// TwinCAT 3 PLC project PLC
// ProgramVersion: 3.1.4024.0
// libraries:
//   Tc2_Standard, * (Beckhoff Automation GmbH)
//   Tc2_System, * (Beckhoff Automation GmbH)
//   Tc3_Module, * (Beckhoff Automation GmbH)
//   Util, * (System)
// project tree:
//   Diagnostic/ GVL_Diagnostic.TcGVL, ST_Diagnostic.TcDUT
//   FLM/Corking/ FB_CorkingRotation.TcPOU, E_FLM_CorkingStep.TcDUT, FB_FLM_CorkingStateMachine.TcPOU, ST_FLM_CorkingParams.TcDUT, ST_FLM_CorkingStatus.TcDUT
//   FLM/Enums/ E_FLM_Step.TcDUT
//   FLM/FBs/ FB_FLM_Diagnostic.TcPOU, FB_FLM_ReadCmd.TcPOU, FB_FLM_ReadCtrl.TcPOU, FB_FLM_ReadInputs.TcPOU, FB_FLM_ResetCmd.TcPOU, FB_FLM_WriteOutputs.TcPOU, FB_FLM_StateMachine.TcPOU
//   FLM/ FB_FLM_Main.TcPOU
//   FLM/Functions/ F_FLM_RawToLevel.TcPOU
//   FLM/Structs/ ST_FLM_Cmd.TcDUT, ST_FLM_Ctrl.TcDUT, ST_FLM_In.TcDUT, ST_FLM_Motion.TcDUT, ST_FLM_Out.TcDUT, ST_FLM_Params.TcDUT, ST_FLM_RawIn.TcDUT, ST_FLM_RawOut.TcDUT, ST_FLM_Status.TcDUT, ST_FLM_StatusSaved.TcDUT
//   / GlobalTextList.TcGTLO, PlcTask.TcTTO, SimuTask.TcTTO, VisualizationManager.TcVMO (not stored)
//   GVLs/ GVL_PLC.TcGVL
//   POUs/ PLC_MAIN.TcPOU, SIMU_MAIN.TcPOU
//   Simulation/ FB_VisuSim.TcPOU
//   StateMachinePro/ E_Step.TcDUT, FB_StateMachinePro.TcPOU
//   StateMachine/ FB_StateMachine.TcPOU
//   VISUs/ Visu.TcVIS
// real-time tasks:
//   TASK PlcTask: cycle T#10ms, priority 20, ADS port 350
//   TASK VISU_TASK: cycle T#200000us, priority 30, ADS port 351
//   TASK SimuTask: cycle T#10ms, priority 21, ADS port 352

CONFIGURATION PLC
    RESOURCE PLC ON TwinCAT3
        TASK PlcTask(INTERVAL := T#10ms, PRIORITY := 20);
        TASK SimuTask(INTERVAL := T#10ms, PRIORITY := 21);
        PROGRAM PLC_MAIN WITH PlcTask : PLC_MAIN;
        PROGRAM SIMU_MAIN WITH SimuTask : SIMU_MAIN;
    END_RESOURCE
END_CONFIGURATION

// ---- Diagnostic/ST_Diagnostic.TcDUT
(* -----------------------------------------------------------------------------
| This sample has been supplied by Beckhoff As-Is and is intended only as an   |
| example implementation. Functionality is not guaranteed.                     |
----------------------------------------------------------------------------- *)

TYPE ST_Diagnostic :
STRUCT
	aCritical : ARRAY[0..GVL_Diagnostic.cMAXEVENTS - 1] OF BOOL;	// eventi critici
	aError : ARRAY[0..GVL_Diagnostic.cMAXEVENTS - 1] OF BOOL;		// errori
	aWarning : ARRAY[0..GVL_Diagnostic.cMAXEVENTS - 1] OF BOOL;		// segnalazioni
	aInfo : ARRAY[0..GVL_Diagnostic.cMAXEVENTS - 1] OF BOOL;		// informazioni
	aVerbose : ARRAY[0..GVL_Diagnostic.cMAXEVENTS - 1] OF BOOL;		// messaggi
END_STRUCT
END_TYPE

// ---- FLM/Enums/E_FLM_Step.TcDUT
(* -----------------------------------------------------------------------------
| This sample has been supplied by Beckhoff As-Is and is intended only as an   |
| example implementation. Functionality is not guaranteed.                     |
----------------------------------------------------------------------------- *)

{attribute 'qualified_only'}
{attribute 'strict'}
{attribute 'to_string'}

TYPE E_FLM_Step :
(
	(* special steps *)
	NoStep := -32767,		// nessuno step
	Unknown := -32000,		// step sconosciuto
	
	(* Error steps *)
	NeOrError := -990,		// non abilitata o in errore
	Reset := -980,			// azzeramento errori

	(* Stop *)
	Stop := 0,				// stop
	
	(* Cycle *)
	Feeding := 110,			// avanzamento
	WaterFilling := 120,	// riempimento acqua
	MintFilling := 130,		// riempimento menta
	Corking := 150,			// tappatura	
		
	(* Stopping *)
	Stopping := 900
	
);
END_TYPE

// ---- FLM/Corking/E_FLM_CorkingStep.TcDUT
(* -----------------------------------------------------------------------------
| This sample has been supplied by Beckhoff As-Is and is intended only as an   |
| example implementation. Functionality is not guaranteed.                     |
----------------------------------------------------------------------------- *)

{attribute 'qualified_only'}
{attribute 'strict'}
{attribute 'to_string'}

TYPE E_FLM_CorkingStep :
(
	(* special steps *)
	NoStep := -32767,		// nessuno step
	Unknown := -32000,		// step sconosciuto
	
	(* Error steps *)
	NeOrError := -990,		// non abilitata o in errore
	Reset := -980,			// azzeramento errori
		
	(* Stop *)
	Stop := 0,
	
	(* Ready *)
	Ready := 100,	
	
	(* Cycle *)
	Down := 200,			// movimento verticale verso il basso
	Rotation := 210,		// rotazione 
	Up := 220,				// movimento verticale verso l'alto
	Done := 230,			// ciclo concluso
	(* Stopping *)
	Stopping := 900	
);
END_TYPE

// ---- FLM/Corking/ST_FLM_CorkingParams.TcDUT
(* -----------------------------------------------------------------------------
| This sample has been supplied by Beckhoff As-Is and is intended only as an   |
| example implementation. Functionality is not guaranteed.                     |
----------------------------------------------------------------------------- *)

TYPE ST_FLM_CorkingParams :
STRUCT
	tDown : TIME := T#1S;			// durata del movimento verso il basso
	tUp : TIME := T#500MS;			// durata movimento verso l'alto	
END_STRUCT
END_TYPE

// ---- FLM/Corking/ST_FLM_CorkingStatus.TcDUT
(* -----------------------------------------------------------------------------
| This sample has been supplied by Beckhoff As-Is and is intended only as an   |
| example implementation. Functionality is not guaranteed.                     |
----------------------------------------------------------------------------- *)

TYPE ST_FLM_CorkingStatus :
STRUCT
	eStep : E_FLM_CorkingStep;				// passo della macchina a stati
	stRstep : STRING;						// passo come stringa
	tStepTime : TIME;						// tempo di permanenza nello stato
	eErrorStep : E_FLM_CorkingStep;			// stato in cui si è generato l'errore
	nErrorID : UDINT;						// id errore
END_STRUCT	
END_TYPE

// ---- FLM/Structs/ST_FLM_Cmd.TcDUT
(* -----------------------------------------------------------------------------
| This sample has been supplied by Beckhoff As-Is and is intended only as an   |
| example implementation. Functionality is not guaranteed.                     |
----------------------------------------------------------------------------- *)

TYPE ST_FLM_Cmd :
STRUCT
	bAck				: BOOL;	(* Riconoscimento allarmi *)
	bStop				: BOOL;	(* Arresta la macchina *)
	bStart				: BOOL;	(* Mette in marcia la macchina *)
END_STRUCT
END_TYPE

// ---- FLM/Structs/ST_FLM_Ctrl.TcDUT
(* -----------------------------------------------------------------------------
| This sample has been supplied by Beckhoff As-Is and is intended only as an   |
| example implementation. Functionality is not guaranteed.                     |
----------------------------------------------------------------------------- *)

TYPE ST_FLM_Ctrl :
STRUCT
	bEmergency: BOOL;	// Emergenza. Deve essere TRUE perchè la macchina possa operare
	bEnable: BOOL;		// Abilitazione macchina. Deve essere TRUE perchè la macchina possa operare
END_STRUCT
END_TYPE

// ---- FLM/Structs/ST_FLM_In.TcDUT
(* -----------------------------------------------------------------------------
| This sample has been supplied by Beckhoff As-Is and is intended only as an   |
| example implementation. Functionality is not guaranteed.                     |
----------------------------------------------------------------------------- *)

TYPE ST_FLM_In :
STRUCT
	(* digital *)
	bEmergency : BOOL;						// emergenza (NC)
	bStartButton : BOOL;					// pulsante di start (NO)
	bStopButton : BOOL;						// pulsante di stop (NO)
	bAckButton : BOOL;						// pulsante di riconoscimento allarmi (NO)
	bBottle : BOOL;							// fotocellula presenza bottiglia (NO)
	bCorkingRotationLimitSwitch : BOOL;		// finecorsa rotazione tappatura (NO)
	(* analog *)
	fWaterLevel : REAL;		// livello acqua
	fMintLevel : REAL;		// livello menta			
END_STRUCT
END_TYPE

// ---- FLM/Structs/ST_FLM_Motion.TcDUT
(* -----------------------------------------------------------------------------
| This sample has been supplied by Beckhoff As-Is and is intended only as an   |
| example implementation. Functionality is not guaranteed.                     |
----------------------------------------------------------------------------- *)

TYPE ST_FLM_Motion :
STRUCT
	// stVAxisMaster : AXIS_REF;
	// stAxis1 : AXIS_REF;
	// stAxis2 : AXIS_REF;
END_STRUCT
END_TYPE

// ---- FLM/Structs/ST_FLM_Out.TcDUT
(* -----------------------------------------------------------------------------
| This sample has been supplied by Beckhoff As-Is and is intended only as an   |
| example implementation. Functionality is not guaranteed.                     |
----------------------------------------------------------------------------- *)

TYPE ST_FLM_Out :
STRUCT
	bFixedYellow : BOOL;		// luce gialla fissa
	bBlinkingYellow: BOOL;		// luce gialla lampeggiante
	bFixedGreen : BOOL;			// luce verde fissa
	bBlinkingGreen : BOOL;		// luce verde lampeggiante
	bHorn : BOOL;				// sirena di segnalazione
	
	bConveyor : BOOL;			// nastro trasportatore
	
	bWater : BOOL;				// riempimento acqua
	bMint : BOOL;				// riempimento menta	
	
	bCorkingVertical : BOOL;	// inserimento del tappo - movimento verticale
	bCorkingRotation : BOOL;	// inserimento del tappo - rotazione
END_STRUCT
END_TYPE

// ---- FLM/Structs/ST_FLM_Params.TcDUT
(* -----------------------------------------------------------------------------
| This sample has been supplied by Beckhoff As-Is and is intended only as an   |
| example implementation. Functionality is not guaranteed.                     |
----------------------------------------------------------------------------- *)

TYPE ST_FLM_Params :
STRUCT
	nFillingCycles : UINT := 3;				// cicli di riempimento
	tWaterFillingTime : TIME := T#1S;		// durata riempimento acqua per ciclo
	tMintFillingTime : TIME := T#500MS;		// durata riempimento menta per ciclo
	fWaterMaxLevel : REAL := 1000.0;		// livello massimo letto dal sensore (acqua)
	fMintMaxLevel : REAL := 200.0;			// livello massimo letto dal sensore (menta)
	stCorking : ST_FLM_CorkingParams;		// parametri dispositivo di tappatura
END_STRUCT
END_TYPE

// ---- FLM/Structs/ST_FLM_RawIn.TcDUT
(* -----------------------------------------------------------------------------
| This sample has been supplied by Beckhoff As-Is and is intended only as an   |
| example implementation. Functionality is not guaranteed.                     |
----------------------------------------------------------------------------- *)

TYPE ST_FLM_RawIn :
STRUCT
	(* digital *)
	bEmergency : BOOL;						// emergenza (NC)
	bStartButton : BOOL;					// pulsante di start (NO)
	bStopButton : BOOL;						// pulsante di stop (NC)
	bAckButton : BOOL;						// pulsante di riconoscimento allarmi (NO)
	bBottle : BOOL;							// fotocellula presenza bottiglia (NO)
	bCorkingRotationLimitSwitch : BOOL;		// finecorsa rotazione tappatura (NO)
	(* analog *)
	nWaterLevel : INT;						// livello acqua
	nMintLevel : INT;						// livello menta
END_STRUCT
END_TYPE

// ---- FLM/Structs/ST_FLM_RawOut.TcDUT
(* -----------------------------------------------------------------------------
| This sample has been supplied by Beckhoff As-Is and is intended only as an   |
| example implementation. Functionality is not guaranteed.                     |
----------------------------------------------------------------------------- *)

TYPE ST_FLM_RawOut :
STRUCT
	bConveyor : BOOL;			// nastro trasportatore
	bWater : BOOL;				// riempimento acqua
	bMint : BOOL;				// riempimento menta	
	bYellow : BOOL;				// luce gialla
	bGreen : BOOL;				// luce verde
	bHorn : BOOL;				// sirena di segnalazione
	bCorkingVertical : BOOL;	// inserimento del tappo - movimento verticale
	bCorkingRotation : BOOL;	// inserimento del tappo - rotazione
END_STRUCT
END_TYPE

// ---- FLM/Structs/ST_FLM_Status.TcDUT
(* -----------------------------------------------------------------------------
| This sample has been supplied by Beckhoff As-Is and is intended only as an   |
| example implementation. Functionality is not guaranteed.                     |
----------------------------------------------------------------------------- *)

TYPE ST_FLM_Status :
STRUCT
	
	stSaved : ST_FLM_StatusSaved;		// Valori ritenuti - utili p.e. per statistiche
	bCritical : BOOL;					// la macchina ha almento una condizione critica attiva
	bError : BOOL;						// la macchina ha almento una condizione di errore attiva	
	bWarning : BOOL;					// la macchina ha almeno una segnalazione attiva	
	bInfo : BOOL;						// la macchina ha almeno una informazione attiva			
	bVerbose : BOOL;					// la macchina ha almeno un messaggio attiva
	
	bFailure : BOOL;					// la macchina è in avaria (critica + error)	
	eStep : E_FLM_Step;					// passo della macchina a stati
	strStep : STRING;					// passo come stringa
	tStepTime : TIME;					// tempo di permanenza nel passo
	eErrorStep : E_FLM_Step;			// passo in cui si è generato l'errore
	nErrorID : DINT;					// codice di erroe
	
	stCorking : ST_FLM_CorkingStatus;	// struttura di stato del dispositivo di tappatura
	
END_STRUCT
END_TYPE

// ---- FLM/Structs/ST_FLM_StatusSaved.TcDUT
(* -----------------------------------------------------------------------------
| This sample has been supplied by Beckhoff As-Is and is intended only as an   |
| example implementation. Functionality is not guaranteed.                     |
----------------------------------------------------------------------------- *)

TYPE ST_FLM_StatusSaved :
STRUCT
	nPowerOnCnt	: UDINT;				// contatore accensioni macchina
	nStartStopCnt : UDINT;				// contatore avvii macchina
	nCCyclesCnt : UDINT;				// contatore cicli di riempimento
	nCriticalCnt : UDINT;				// contatore eventi critici
	nErrorCnt : UDINT;					// contatore errori	
	nWarningCnt : UDINT;				// contatore segnalazioni
END_STRUCT
END_TYPE

// ---- StateMachinePro/E_Step.TcDUT
{attribute 'qualified_only'}
{attribute 'strict'}
{attribute 'to_string'}

TYPE E_Step :
(
	(* special steps *)
	NoStep := -32767,		// nessuno step
	Unknown := -32000,		// step sconosciuto
	
	(* Not Enabled or Errors*)
	NeOrError := -990,			// non abilitata o in errore

	(* Stop *)
	Stop := 0,				// stop
	
	(* Preparation *)
	Feeding := 110,			// avanzamento
	WaterFilling := 120,	// riempimento acqua
	MintFilling := 130,		// riempimento menta
	Waiting1 := 140,		// attesa 1
	Corking := 150,			// tappatura
	Waiting2 := 160,		// attesa 2
		
	(* Stopping *)
	Stopping := 900
	
);
END_TYPE

// ---- Diagnostic/GVL_Diagnostic.TcGVL
(* -----------------------------------------------------------------------------
| This sample has been supplied by Beckhoff As-Is and is intended only as an   |
| example implementation. Functionality is not guaranteed.                     |
----------------------------------------------------------------------------- *)

{attribute 'qualified_only'}
VAR_GLOBAL CONSTANT
	cMAXEVENTS : UDINT := 64;
END_VAR

// ---- GVLs/GVL_PLC.TcGVL
(* -----------------------------------------------------------------------------
| This sample has been supplied by Beckhoff As-Is and is intended only as an   |
| example implementation. Functionality is not guaranteed.                     |
----------------------------------------------------------------------------- *)

{attribute 'qualified_only'}
VAR_GLOBAL PERSISTENT	
	stFlmParams : ST_FLM_Params;
	stFlmStatusSaved : ST_FLM_StatusSaved;
END_VAR

VAR_GLOBAL
	stFlmDiagnostic	: ST_Diagnostic;

	stFlmIn : ST_FLM_In;
	stFlmRawIn : ST_FLM_RawIn;
	stFlmOut : ST_FLM_Out;
	stFlmRawOut : ST_FLM_RawOut;
	stFlmCtrl : ST_FLM_Ctrl;	
	stFlmStatus : ST_FLM_Status;
	stFlmMotion	: ST_FLM_Motion;

END_VAR

// ---- POUs/PLC_MAIN.TcPOU
(* -----------------------------------------------------------------------------
| This sample has been supplied by Beckhoff As-Is and is intended only as an   |
| example implementation. Functionality is not guaranteed.                     |
----------------------------------------------------------------------------- *)

PROGRAM PLC_MAIN
VAR
	bInitialized : BOOL;
	
	fbGetCurTaskIndex : GETCURTASKINDEX;		
	tTaskCycleTime : UDINT;					// tempo di ciclo della task in microsecondi
	tTaskExecTime : UDINT;					// tempo di esecuzione della task in microsecondi
	tTaskMaxExecTime : UDINT;				// tempo massimo di esecuzione della task in microsecondi

	fbFlm : FB_FLM_Main;
	
	
	// fbTest : FB_FLM_CorkingStateMachine;
END_VAR

(* -----------------------------------------------------------------------------
| This sample has been supplied by Beckhoff As-Is and is intended only as an   |
| example implementation. Functionality is not guaranteed.                     |
----------------------------------------------------------------------------- *)

IF NOT bInitialized THEN
	
	// Get the Cycle Time of the task to which this PRG is assigned (it will then be shared with the State Machine)
	fbGetCurTaskIndex();
	tTaskCycleTime := _TaskInfo[fbGetCurTaskIndex.index].CycleTime / 10;	// CycleTime is expressed in multiples of 100ns
	bInitialized := TRUE;
	
ELSE
	
	(* task time *)
	tTaskExecTime := _TaskInfo[fbGetCurTaskIndex.index].LastExecTime / 10;		// ExecTime is expressed in multiples of 100ns
	IF tTaskExecTime > tTaskMaxExecTime THEN
			tTaskMaxExecTime := tTaskExecTime;
	END_IF;	
	
	(* machine *)
		
	fbFlm(
		bEnable:= TRUE, 
		tTaskCycleTime:= tTaskCycleTime, 
		nId:= 0, 
		bHwError:= FALSE,	
		stRawIn := GVL_PLC.stFlmRawIn,
		stIn := GVL_PLC.stFlmIn,
		stRawOut := GVL_PLC.stFlmRawOut,
		stOut := GVL_PLC.stFlmOut,
		stCtrl := GVL_PLC.stFlmCtrl,		
		stParams := GVL_PLC.stFlmParams,
		stDiagnostic := GVL_PLC.stFlmDiagnostic,
		stStatus := GVL_PLC.stFlmStatus,
		stStatusSaved := GVL_PLC.stFlmStatusSaved,
		stMotion := GVL_PLC.stFlmMotion,	 
	);
		
	
		
	(* 
	fbTest(
		bEnable:= TRUE, 
		bAck:= GVL_PLC.stFlmIn.bAckButton, 
		bStart:= GVL_PLC.stFlmIn.bStartButton, 
		bStop:= GVL_PLC.stFlmIn.bStopButton, 
		bRotationLimitSwitch:= GVL_PLC.stFlmIn.bCorkingRotationLimitSwitch, 
		stParams:= GVL_PLC.stFlmParams.stCorking, 
	);
	*)
END_IF

END_PROGRAM

// ---- FLM/FB_FLM_Main.TcPOU
(* -----------------------------------------------------------------------------
| This sample has been supplied by Beckhoff As-Is and is intended only as an   |
| example implementation. Functionality is not guaranteed.                     |
----------------------------------------------------------------------------- *)

FUNCTION_BLOCK FB_FLM_Main

VAR_INPUT
	bEnable			: BOOL;
	tTaskCycleTime	: UDINT;
	nId				: USINT;	
	bHwError		: BOOL;	
END_VAR

VAR_OUTPUT

END_VAR
	
VAR_IN_OUT
	stRawIn : ST_FLM_RawIn;
	stIn : ST_FLM_In;	
	stRawOut : ST_FLM_RawOut;
	stOut : ST_FLM_Out;
	stCtrl : ST_FLM_Ctrl;	
	stParams : ST_FLM_Params;
	stDiagnostic : ST_Diagnostic;
	stStatus : ST_FLM_Status;
	stStatusSaved : ST_FLM_StatusSaved;
	stMotion : ST_FLM_Motion;

END_VAR

VAR
	bInitialized : BOOL;
	stCmd : ST_FLM_Cmd;
	errno : INT;
	(* fbReadPar : fbMachineReadPars; *)
	fbReadCmd : FB_FLM_ReadCmd;
	fbResetCmd : FB_FLM_ResetCmd;
	fbReadCtrl : FB_FLM_ReadCtrl;
	fbReadIn : FB_FLM_ReadInputs;
	fbDiagnostic : FB_FLM_Diagnostic;
	fbStateMachine : FB_FLM_StateMachine;
	fbCorkingStateMachine : FB_FLM_CorkingStateMachine;
	
	fbWriteOut : FB_FLM_WriteOutputs;
	
END_VAR

(* -----------------------------------------------------------------------------
| This sample has been supplied by Beckhoff As-Is and is intended only as an   |
| example implementation. Functionality is not guaranteed.                     |
----------------------------------------------------------------------------- *)

IF NOT bInitialized THEN
	stStatus.stSaved := stStatusSaved;
	bInitialized := TRUE;		
ELSE

	(* 01 - Leggi ingressi, controlli, parametri e comandi  *)	
	fbReadIn(
		stParams := stParams,		
		stRawIn := stRawIn
	);				
	
	stIn := fbReadIn.stIn;
	fbReadCtrl(
		nId := nId,	
		bEnable := bEnable,
		stIn := stIn,	
				
	);
	stCtrl := fbReadCtrl.stCtrl;
		
	fbReadCmd(stIn := stIn);
	stCmd := fbReadCmd.stCmd;	

	(* 03 - Gestione eventi *)	
	fbDiagnostic(
		stIn := stIn,
		stOut := stOut,
		stCtrl := stCtrl,
		stParams := stParams,
		bHwError := bHwError, 
		bAck := stCmd.bAck, 
		stStatus := stStatus, 
		stMotion := stMotion,
		stDiagnostic := stDiagnostic, 
	);
	stStatus.bCritical := fbDiagnostic.bCritical;
	stStatus.bError := fbDiagnostic.bError;
	stStatus.bWarning := fbDiagnostic.bWarning;
	stStatus.bInfo := fbDiagnostic.bInfo;
	stStatus.bVerbose := fbDiagnostic.bVerbose;
	stStatus.bFailure := fbDiagnostic.bFailure;
	
	stOut.bBlinkingYellow := fbDiagnostic.bBlinking;
	stOut.bFixedYellow := fbDiagnostic.bFixed;
	stOut.bHorn := fbDiagnostic.bHorn;

	(* 04 - Macchina a stati principale: *)		
	fbStateMachine(
		stIn := stIn,
		stCtrl := stCtrl,
		StCmd := stCmd,
		stParams := stParams,
		stStatus := stStatus,		
	);	
	stStatus.eStep := fbStateMachine.eStep;
	stStatus.strStep := TO_STRING(stStatus.eStep);
	stStatus.tStepTime := fbStateMachine.tStepTime;
	stStatus.eErrorStep := fbStateMachine.eErRstep; 
	stStatus.nErrorID := fbStateMachine.nErrId;
	
	stOut.bConveyor := fbStateMachine.bConveyor;
	stOut.bWater := fbStateMachine.bWater;
	stOut.bMint := fbStateMachine.bMint;
	stOut.bBlinkingGreen := fbStateMachine.bBlinkingGreen;
	stOut.bFixedGreen := fbStateMachine.bFixedGreen;
	
	(* 05 - Macchine a stati secondarie *)
	fbCorkingStateMachine(
		bEnable:= stCtrl.bEnable AND stCtrl.bEmergency AND NOT stStatus.bFailure,
		bAck:= stCmd.bAck, 
		bStart:= fbStateMachine.bCorkingStart, 
		bStop:= stCmd.bStop, 
		bRotationLimitSwitch:= stIn.bCorkingRotationLimitSwitch, 
		stParams:= stParams.stCorking,		 
	);
	stStatus.stCorking.eStep := fbCorkingStateMachine.eStep;
	stStatus.stCorking.tStepTime := fbCorkingStateMachine.tStepTime;
	stStatus.stCorking.eErrorStep := fbCorkingStateMachine.eErrStep;
	stStatus.stCorking.nErrorID	:= fbCorkingStateMachine.nErrID; 
	
	stOut.bCorkingRotation := fbCorkingStateMachine.bRotation;
	stOut.bCorkingVertical := fbCorkingStateMachine.bVertical;
	
	(* 06 - Scrivi uscite e informazioni *)	
	fbWriteOut(		
		stOut		:= stOut,
		stParams	:= stParams,		
		stRawOut	:= stRawOut
	);
	
	// stStatus.stSaved.nCounter := stStatus.stSaved.nCounter +1;	   
	
	stStatusSaved := stStatus.stSaved;		// aggiorna struttura con i dati salvati

	(* 07 - fine - altre operazioni*)
		
	fbResetCmd();

END_IF;

END_FUNCTION_BLOCK

// ---- FLM/FBs/FB_FLM_ReadCmd.TcPOU
(* -----------------------------------------------------------------------------
| This sample has been supplied by Beckhoff As-Is and is intended only as an   |
| example implementation. Functionality is not guaranteed.                     |
----------------------------------------------------------------------------- *)

FUNCTION_BLOCK FB_FLM_ReadCmd

VAR_INPUT
	stIn : ST_FLM_In;
END_VAR

VAR_OUTPUT
	stCmd : ST_FLM_Cmd;
END_VAR

VAR_IN_OUT
	
END_VAR

VAR
	fbRtStart	: R_TRIG;
	fbRtStop	: R_TRIG;
	fbTpAck		: TP;	
END_VAR
VAR CONSTANT
	
END_VAR

(* -----------------------------------------------------------------------------
| This sample has been supplied by Beckhoff As-Is and is intended only as an   |
| example implementation. Functionality is not guaranteed.                     |
----------------------------------------------------------------------------- *)

fbRtStart(	CLK := stIn.bStartButton);
fbRtStop(	CLK := stIn.bStopButton);
fbTpAck(IN:= stIn.bAckButton, PT:= T#200MS);


stCmd.bAck		:= fbTpAck.Q;
stCmd.bStop		:= fbRtStop.Q;
stCmd.bStart	:= fbRtStart.Q;

END_FUNCTION_BLOCK

// ---- FLM/FBs/FB_FLM_ResetCmd.TcPOU
(* -----------------------------------------------------------------------------
| This sample has been supplied by Beckhoff As-Is and is intended only as an   |
| example implementation. Functionality is not guaranteed.                     |
----------------------------------------------------------------------------- *)

FUNCTION_BLOCK FB_FLM_ResetCmd

VAR_INPUT

END_VAR

VAR_IN_OUT
	
END_VAR

VAR
	
END_VAR

(* -----------------------------------------------------------------------------
| This sample has been supplied by Beckhoff As-Is and is intended only as an   |
| example implementation. Functionality is not guaranteed.                     |
----------------------------------------------------------------------------- *)

;

END_FUNCTION_BLOCK

// ---- FLM/FBs/FB_FLM_ReadCtrl.TcPOU
(* -----------------------------------------------------------------------------
| This sample has been supplied by Beckhoff As-Is and is intended only as an   |
| example implementation. Functionality is not guaranteed.                     |
----------------------------------------------------------------------------- *)

FUNCTION_BLOCK FB_FLM_ReadCtrl

VAR_INPUT
	nId:	INT;
	bEnable : BOOL;
	stIn : ST_FLM_In;
END_VAR

VAR_OUTPUT
	stCtrl : ST_FLM_Ctrl;
END_VAR

VAR
	fbTonStartup: TON;
END_VAR

(* -----------------------------------------------------------------------------
| This sample has been supplied by Beckhoff As-Is and is intended only as an   |
| example implementation. Functionality is not guaranteed.                     |
----------------------------------------------------------------------------- *)

fbTonStartup(IN := TRUE, PT := T#3S);
stCtrl.bEmergency := stIn.bEmergency;
stCtrl.bEnable := fbTonStartup.Q AND bEnable;

END_FUNCTION_BLOCK

// ---- FLM/FBs/FB_FLM_ReadInputs.TcPOU
(* -----------------------------------------------------------------------------
| This sample has been supplied by Beckhoff As-Is and is intended only as an   |
| example implementation. Functionality is not guaranteed.                     |
----------------------------------------------------------------------------- *)

FUNCTION_BLOCK FB_FLM_ReadInputs

VAR_INPUT
	stParams : ST_FLM_Params;
END_VAR

VAR_IN_OUT	
	stRawIn : ST_FLM_RawIn;
END_VAR

VAR_OUTPUT
	stIn :  ST_FLM_In;
END_VAR

(* -----------------------------------------------------------------------------
| This sample has been supplied by Beckhoff As-Is and is intended only as an   |
| example implementation. Functionality is not guaranteed.                     |
----------------------------------------------------------------------------- *)

(* digital *)
stIn.bEmergency := stRawIn.bEmergency;
stIn.bStartButton := stRawIn.bStartButton;
stIn.bStopButton := NOT stRawIn.bStopButton;
stIn.bAckButton := stRawIn.bAckButton;
stIn.bBottle := stRawIn.bBottle;
stIn.bCorkingRotationLimitSwitch := stRawIn.bCorkingRotationLimitSwitch;

(* analog *)
stIn.fWaterLevel := F_FLM_RawToLevel(stRawIn.nWaterLevel, stParams.fWaterMaxLevel);
stIn.fMintLevel := F_FLM_RawToLevel(stRawIn.nMintLevel, stParams.fMintMaxLevel);

END_FUNCTION_BLOCK

// ---- FLM/Functions/F_FLM_RawToLevel.TcPOU
(* -----------------------------------------------------------------------------
| This sample has been supplied by Beckhoff As-Is and is intended only as an   |
| example implementation. Functionality is not guaranteed.                     |
----------------------------------------------------------------------------- *)

FUNCTION F_FLM_RawToLevel : REAL
VAR_INPUT
	nRaw : INT;			// valore letto dagli ingressi	
	rMaxLevel : REAL;
END_VAR
VAR_OUTPUT
    fLevel : REAL;		// [mm]	Livello
END_VAR
VAR
	
END_VAR
VAR CONSTANT
	cMAXRAW : INT := 2#0111_1111_1111_1111;	// massimo valore ingresso analogico
END_VAR

(* -----------------------------------------------------------------------------
| This sample has been supplied by Beckhoff As-Is and is intended only as an   |
| example implementation. Functionality is not guaranteed.                     |
----------------------------------------------------------------------------- *)

F_FLM_RawToLevel := (TO_REAL(nRaw) / TO_REAL(cMAXRAW)) * rMaxLevel;

END_FUNCTION

// ---- FLM/FBs/FB_FLM_Diagnostic.TcPOU
(* -----------------------------------------------------------------------------
| This sample has been supplied by Beckhoff As-Is and is intended only as an   |
| example implementation. Functionality is not guaranteed.                     |
----------------------------------------------------------------------------- *)

FUNCTION_BLOCK FB_FLM_Diagnostic
VAR_INPUT
	stIn : ST_FLM_In;
	stOut : ST_FLM_Out;
	stParams : ST_FLM_Params;
	stCtrl : ST_FLM_Ctrl;
	bHwError : BOOL;
	bAck : BOOL;
	stStatus : ST_FLM_Status;
END_VAR

VAR_IN_OUT
	stMotion : ST_FLM_Motion;
	stDiagnostic : ST_Diagnostic;
END_VAR

VAR_OUTPUT	
	bCritical : BOOL;
	bError : BOOL;
	bWarning : BOOL;
	bInfo  : BOOL;
	bVerbose : BOOL;
	bFailure : BOOL;
	bBlinking : BOOL;
	bFixed : BOOL;
	bHorn : BOOL;
END_VAR

VAR	
	stInstantDiagnostic : ST_Diagnostic;	
	nUi : UDINT;

END_VAR

(* -----------------------------------------------------------------------------
| This sample has been supplied by Beckhoff As-Is and is intended only as an   |
| example implementation. Functionality is not guaranteed.                     |
----------------------------------------------------------------------------- *)

(* reSet condizioni istantantanee *)
FOR nUi := 0 TO GVL_Diagnostic.cMAXEVENTS -1 DO
	stInstantDiagnostic.aCritical[nUi]	:= 0;
	stInstantDiagnostic.aError[nUi]		:= 0;
	stInstantDiagnostic.aWarning[nUi]	:= 0;
	stInstantDiagnostic.aInfo[nUi]		:= 0;
	stInstantDiagnostic.aVerbose[nUi]	:= 0; 
END_FOR

(* filtri, etc *)

(* imposta condizioni istantanee *)
stInstantDiagnostic.aCritical[0] := bHwError;
stInstantDiagnostic.aCritical[1] := NOT stCtrl.bEmergency;

stInstantDiagnostic.aError[0] := stStatus.eErrorStep <> E_FLM_Step.NoStep;
stInstantDiagnostic.aError[1] := stStatus.stCorking.eErrorStep <> E_FLM_CorkingStep.NoStep;
stInstantDiagnostic.aError[2] := (stStatus.eStep > E_FLM_Step.Stop) AND (stIn.fWaterLevel < stParams.fWaterMaxLevel * 0.1);
stInstantDiagnostic.aError[3] := (stStatus.eStep > E_FLM_Step.Stop) AND (stIn.fMintLevel < stParams.fMintMaxLevel * 0.1);

stInstantDiagnostic.aWarning[0] := (stStatus.eStep > E_FLM_Step.Stop) AND (stIn.fWaterLevel < stParams.fWaterMaxLevel * 0.3);
stInstantDiagnostic.aWarning[1] := (stStatus.eStep > E_FLM_Step.Stop) AND (stIn.fMintLevel < stParams.fMintMaxLevel * 0.3);

(* reset condizioni ritenute *)
IF bAck THEN
	FOR nUi := 0 TO GVL_Diagnostic.cMAXEVENTS -1 DO
		stDiagnostic.aCritical[nUi] := 0;
		stDiagnostic.aError[nUi] := 0;
		stDiagnostic.aWarning[nUi] := 0;
		stDiagnostic.aInfo[nUi] := 0;
		stDiagnostic.aVerbose[nUi] := 0; 
	END_FOR
	bCritical := FALSE;
	bError := FALSE;
	bWarning := FALSE;
	bInfo := FALSE;
	bVerbose := FALSE;
	bBlinking := FALSE;
	bHorn := FALSE;
END_IF									

(* imposta condizioni ritenute *)									
FOR nUi := 0 TO GVL_Diagnostic.cMAXEVENTS -1 DO
	IF stInstantDiagnostic.aCritical[nUi] THEN
		stDiagnostic.aCritical[nUi] := TRUE;
		bCritical := TRUE;
	END_IF
	IF stInstantDiagnostic.aError[nUi] THEN
		stDiagnostic.aError[nUi] := TRUE;
		bError := TRUE;
	END_IF
	IF stInstantDiagnostic.aWarning[nUi] THEN
		stDiagnostic.aWarning[nUi] := TRUE;
		bWarning := TRUE;
	END_IF
	IF stInstantDiagnostic.aInfo[nUi] THEN
		stDiagnostic.aInfo[nUi] := TRUE;
		bInfo := TRUE;
	END_IF
	IF stInstantDiagnostic.aVerbose[nUi] THEN
		stDiagnostic.aVerbose[nUi] := TRUE;
		bVerbose := TRUE;
	END_IF
END_FOR

bFailure := bCritical OR bError;

bBlinking := bFailure;
bHorn := bFailure;
bFixed := bWarning;

END_FUNCTION_BLOCK

// ---- FLM/FBs/FB_FLM_StateMachine.TcPOU
(* -----------------------------------------------------------------------------
| This sample has been supplied by Beckhoff As-Is and is intended only as an   |
| example implementation. Functionality is not guaranteed.                     |
----------------------------------------------------------------------------- *)

FUNCTION_BLOCK FB_FLM_StateMachine
VAR_INPUT	
	stIn		: ST_FLM_In;
	stCtrl		: ST_FLM_Ctrl;
	stCmd		: ST_FLM_Cmd;
	stParams	: ST_FLM_Params;
	stStatus	: ST_FLM_Status;
END_VAR

VAR_OUTPUT
	eStep :  E_FLM_Step;
	tStepTime : TIME;
	eErrStep : E_FLM_Step;
	nErrId : DINT;
	
	bConveyor : BOOL;			// nastro trasportatore
	bWater : BOOL;				// riempimento acqua
	bMint : BOOL;				// riempimento menta	
	bCorkingStart : BOOL;		// start inserimento del tappo	
	bBlinkingGreen : BOOL;		// lampada verde lampeggiante
	bFixedGreen : BOOL;			// lampada verde lampeggiante
END_VAR

VAR_IN_OUT
	
END_VAR

VAR
	bInitialized :  BOOL;
	eNewstep :  E_FLM_Step;
	bEntryact :  BOOL;
	fbTonStep :  TON;	
	
	fbTonBottle : TON;
	fbRtBottle : R_TRIG;
		
	bStopRequest : BOOL;
	
	nFillingCycles : USINT;
END_VAR

(* -----------------------------------------------------------------------------
| This sample has been supplied by Beckhoff As-Is and is intended only as an   |
| example implementation. Functionality is not guaranteed.                     |
----------------------------------------------------------------------------- *)

IF NOT bInitialized THEN
	eNewstep := E_FLM_Step.NoStep;
	eStep := E_FLM_Step.Stop;
	bEntryact := FALSE;
	bInitialized := TRUE;		
ELSE	
	(* disabilitata o avaria *)	
	IF NOT stCtrl.bEnable OR NOT(stCtrl.bEmergency) OR stStatus.bFailure THEN
		eNewstep := E_FLM_Step.NeOrError;
	END_IF
	
	IF eNewstep <> E_FLM_Step.NoStep THEN
		eStep := eNewstep;
		eNewstep := E_FLM_Step.NoStep;
		bEntryact := FALSE;
	END_IF;

	(* filtri *)
	fbTonBottle(IN:= stIn.bBottle, PT:= T#500MS);		// filtro sensore presenza bottiglia
	
	(* fronti *)
	fbRtBottle(CLK:= fbTonBottle.Q);
	
	(* richieste *)
	IF stCmd.bStop THEN
		bStopRequest := TRUE;
	END_IF; 
	
	CASE eStep OF
		
		(* not Enabled or Error *)
		E_FLM_Step.NeOrError :
			(* entry action *)
			IF NOT bEntryact THEN
				bEntryact := TRUE;
			END_IF;

			(* body *)
			bConveyor := FALSE;
			bWater := FALSE;
			bMint := FALSE;
			bCorkingStart := FALSE;
			bBlinkingGreen := FALSE;
			bFixedGreen := FALSE;
			
			nFillingCycles := 0;
					
			(* transition *)
			IF stCtrl.bEnable THEN				
				IF stCmd.bAck THEN
					eNewstep := E_FLM_Step.Reset;
				END_IF
			END_IF

			(* exitact *)
			IF eNewstep <> E_FLM_Step.NoStep THEN
				nErrId := 0;
				eErrStep := E_FLM_Step.NoStep;
			END_IF;

		(* Reset *)
		E_FLM_Step.Reset :
			(* entry action *)
			IF NOT bEntryact THEN				
				bEntryact := TRUE;
			END_IF;

			(* body *)
			bConveyor := FALSE;
			bWater := FALSE;
			bMint := FALSE;
			bCorkingStart := FALSE;
			bBlinkingGreen := FALSE;
			bFixedGreen := FALSE;
			
			nFillingCycles := 0;
					
			(* transition *)
			IF stCtrl.bEnable THEN				
				IF NOT stStatus.bFailure AND stStatus.stCorking.eStep = E_FLM_CorkingStep.Stop THEN
					eNewstep := E_FLM_Step.Stop;
				END_IF
			END_IF

			(* exitact *)
			IF eNewstep <> E_FLM_Step.NoStep THEN
				;
			END_IF;		
			
		(* Stop *)
		E_FLM_Step.Stop:
			(* entry action *)
			IF NOT bEntryact THEN
				bStopRequest := FALSE;
				bEntryact := TRUE;
			END_IF;

			(* body *)
			bConveyor := FALSE;
			bWater := FALSE;
			bMint := FALSE;
			bCorkingStart := FALSE;
			bBlinkingGreen := FALSE;
			bFixedGreen := FALSE;
			
			nFillingCycles := 0;
				
			(* transition *)			
			IF NOT stCmd.bStop AND stCmd.bStart THEN
				eNewstep := E_FLM_Step.Feeding;
			END_IF
			
			(* exitact *)
			IF eNewstep <> E_FLM_Step.NoStep THEN
				;
			END_IF;
			
		(* Feeding *)
		E_FLM_Step.Feeding:
			(* entry action *)
			IF NOT bEntryact THEN
				bEntryact := TRUE;
			END_IF;

			(* body *)
			bConveyor := TRUE;
			bWater := FALSE;
			bMint := FALSE;
			bCorkingStart := FALSE;
			bBlinkingGreen := FALSE;
			bFixedGreen := TRUE;
			bBlinkingGreen := bStopRequest;
			bFixedGreen := TRUE;
		
			(* transition *)
			IF bStopRequest AND NOT stIn.bBottle THEN
				eNewstep := E_FLM_Step.Stopping;
			ELSE
				IF fbRtBottle.Q THEN
					eNewstep := E_FLM_Step.WaterFilling;
				END_IF
			END_IF
			
			(* exitact *)
			IF eNewstep <> E_FLM_Step.NoStep THEN
				;
			END_IF;
			
		(* Water Filling *)
		E_FLM_Step.WaterFilling:
			(* entry action *)
			IF NOT bEntryact THEN
				nFillingCycles := nFillingCycles + 1;
				bEntryact := TRUE;
			END_IF;

			(* body *)
			bConveyor := FALSE;
			bWater := TRUE;
			bMint := FALSE;
			bCorkingStart := FALSE;
			bBlinkingGreen := bStopRequest;
			bFixedGreen := TRUE;
		
			(* transition *)
			IF tStepTime >= stParams.tWaterFillingTime THEN
				eNewstep := E_FLM_Step.MintFilling;
			END_IF
			
			(* exitact *)
			IF eNewstep <> E_FLM_Step.NoStep THEN
				;
			END_IF;
			
		(* Mint Filling *)
		E_FLM_Step.MintFilling:
			(* entry action *)
			IF NOT bEntryact THEN
				bEntryact := TRUE;
			END_IF;

			(* body *)
			bConveyor := FALSE;
			bWater := FALSE;
			bMint := TRUE;
			bCorkingStart := FALSE;
			bBlinkingGreen := bStopRequest;
			bFixedGreen := TRUE;
		
			(* transition *)
			IF tStepTime >= stParams.tMintFillingTime THEN
				IF nFillingCycles >= stParams.nFillingCycles THEN
					eNewstep := E_FLM_Step.Corking;
				ELSE 
					eNewstep := E_FLM_Step.WaterFilling;
				END_IF
					
			END_IF
			
			(* exitact *)
			IF eNewstep <> E_FLM_Step.NoStep THEN
				IF eNewstep = E_FLM_Step.Corking THEN
					nFillingCycles := 0;
				END_IF
			END_IF;	

		(* Corking *)
		E_FLM_Step.Corking:
			(* entry action *)
			IF NOT bEntryact THEN
				bEntryact := TRUE;
			END_IF;

			(* body *)
			bConveyor := FALSE;
			bWater := FALSE;
			bMint := FALSE;
			bCorkingStart := TRUE;
			bBlinkingGreen := bStopRequest;
			bFixedGreen := TRUE;
		
			(* transition *)
			IF stStatus.stCorking.eStep = E_FLM_CorkingStep.Done THEN
				eNewstep := E_FLM_Step.Feeding;
			END_IF
			
			(* exitact *)
			IF eNewstep <> E_FLM_Step.NoStep THEN
				;
			END_IF;

		(* Stopping *)
		E_FLM_Step.Stopping:
			(* entry action *)
			IF NOT bEntryact THEN
				bEntryact := TRUE;
			END_IF;

			(* body *)
			bConveyor := tStepTime < T#500MS;
			bWater := tStepTime >= T#1000MS AND tStepTime <= T#1300MS;
			bMint := tStepTime >= T#1000MS AND tStepTime <= T#1300MS;
			bCorkingStart := FALSE;
			bBlinkingGreen := TRUE;
			bFixedGreen := FALSE;
		
			(* transition *)
			IF tStepTime >= T#4S THEN
				eNewstep := E_FLM_Step.Stop;
			END_IF; 
			
			(* exitact *)
			IF eNewstep <> E_FLM_Step.NoStep THEN
				;
			END_IF;		
		ELSE
			eNewstep := E_FLM_Step.NeOrError;
			eErrStep := E_FLM_Step.Unknown;
			nErrId := -9;			
	END_CASE;
	
	(* tempo di permanenza nello step *)
	fbTonStep(IN := (eNewstep = E_FLM_Step.NoStep), PT := T#500H);
	tStepTime := fbTonStep.ET;
	
END_IF;

END_FUNCTION_BLOCK

// ---- FLM/Corking/FB_FLM_CorkingStateMachine.TcPOU
(* -----------------------------------------------------------------------------
| This sample has been supplied by Beckhoff As-Is and is intended only as an   |
| example implementation. Functionality is not guaranteed.                     |
----------------------------------------------------------------------------- *)

FUNCTION_BLOCK FB_FLM_CorkingStateMachine
VAR_INPUT
	bEnable : BOOL;
	bAck : BOOL;
	bStart : BOOL;
	bStop : BOOL;
	bRotationLimitSwitch : BOOL;
	stParams : ST_FLM_CorkingParams;
END_VAR

VAR_IN_OUT	
	
END_VAR

VAR_OUTPUT
	eStep :  E_FLM_CorkingStep;
	tStepTime :  TIME;
	eErrStep :  E_FLM_CorkingStep;
	nErrID : UDINT;
	bErr : BOOL;
	bVertical : BOOL;
	bRotation : BOOL;
END_VAR

VAR
	bInitialized :  BOOL;
	eNewstep :   E_FLM_CorkingStep;
	bEntryact :  BOOL;
	fbTonStep :  TON;
	ui : UINT;	
	
	fbRtStart : R_TRIG;
	fbRtStop : R_TRIG;
	bStopRequest : BOOL;
	fbRotation : FB_CorkingRotation;
	
	bRotationExecute : BOOL;	
	
	
END_VAR

(* -----------------------------------------------------------------------------
| This sample has been supplied by Beckhoff As-Is and is intended only as an   |
| example implementation. Functionality is not guaranteed.                     |
----------------------------------------------------------------------------- *)

IF NOT bInitialized THEN
	eNewstep :=  E_FLM_CorkingStep.NoStep;
	eStep :=  E_FLM_CorkingStep.Stop;
	bEntryact := FALSE;
	bInitialized := TRUE;	
	bErr := FALSE;
	eErrStep :=  E_FLM_CorkingStep.NoStep;	
	nErrID := 0;	
ELSE	
	
	(* fronti *)
	fbRtStart(CLK:= bStart);
	fbRtStop(CLK:= bStop);	
	
	(* richieste *)
	IF fbRtStop.Q THEN
		bStopRequest := TRUE;
	END_IF; 

	(* disabilitata o avaria *)
	IF NOT bEnable THEN
		eNewstep := E_FLM_CorkingStep.NeOrError;
	END_IF;
	
	IF eNewstep <>  E_FLM_CorkingStep.NoStep THEN
		eStep := eNewstep;
		eNewstep :=  E_FLM_CorkingStep.NoStep;
		bEntryact := FALSE;
	END_IF;

	CASE eStep OF
		(* not Enabled *)
		 E_FLM_CorkingStep.NeOrError :
			(* entry action *)
			IF NOT bEntryact THEN
				bEntryact := TRUE;
			END_IF;

			(* body *)
			bErr := TRUE;
			
			bVertical := FALSE;
			bRotation := FALSE;			
			bRotationExecute := FALSE;			
					
			(* transition *)
			IF bAck THEN
				eNewstep :=  E_FLM_CorkingStep.Reset;								
			END_IF;

			(* exitact *)
			IF eNewstep <>  E_FLM_CorkingStep.NoStep THEN
				nErrID := 0;
				eErrStep := E_FLM_CorkingStep.NoStep;			
			END_IF;	

		(* Reset *)
		E_FLM_CorkingStep.Reset :
			(* entry action *)
			IF NOT bEntryact THEN				
				bEntryact := TRUE;
			END_IF;

			(* body *)
			bErr := FALSE;
			
			bVertical := FALSE;
			bRotation := FALSE;			
			bRotationExecute := FALSE;			
					
			(* transition *)
			IF TRUE THEN
				eNewstep :=  E_FLM_CorkingStep.Stop;
			END_IF
						
			(* exitact *)
			IF eNewstep <>  E_FLM_CorkingStep.NoStep THEN
				;			
			END_IF;
		
		(* Stop *)
		E_FLM_CorkingStep.Stop:
			(* entry action *)
			IF NOT bEntryact THEN
				bStopRequest := FALSE;
				bEntryact := TRUE;
			END_IF;

			(* body *)
			bErr := FALSE;
			
			bVertical := FALSE;
			bRotation := FALSE;			
			bRotationExecute := FALSE;				
							
			(* transition *)
			IF tStepTime > T#1S THEN
				eNewstep :=  E_FLM_CorkingStep.Ready;
			END_IF;

			(* exitact *)
			IF eNewstep <>  E_FLM_CorkingStep.NoStep THEN
				;
			END_IF;
		
		(* Ready *)
		E_FLM_CorkingStep.Ready:
			(* entry action *)
			IF NOT bEntryact THEN
				bEntryact := TRUE;
			END_IF;

			(* body *)
			bErr := FALSE;
			
			bVertical := FALSE;
			bRotation := FALSE;			
			bRotationExecute := FALSE;					
							
			(* transition *)
			IF NOT bStopRequest THEN
				IF NOT bStop AND fbRtStart.Q THEN
					eNewstep :=  E_FLM_CorkingStep.Down;			
				END_IF;
			ELSE
				eNewstep :=  E_FLM_CorkingStep.Stop;
			END_IF

			(* exitact *)
			IF eNewstep <>  E_FLM_CorkingStep.NoStep THEN
				;
			END_IF;
						
		(* Down *)
		E_FLM_CorkingStep.Down:
			(* entry action *)
			IF NOT bEntryact THEN
				bEntryact := TRUE;
			END_IF;

			(* body *)
			bErr := FALSE;
			
			bVertical := TRUE;
			bRotation := FALSE;			
			bRotationExecute := FALSE;					
							
			(* transition *)
			IF NOT bStop THEN
				IF tstepTime >= stParams.tDown THEN
					eNewstep :=  E_FLM_CorkingStep.Rotation;			
				END_IF;
			ELSE
				eNewstep :=  E_FLM_CorkingStep.Stop;
			END_IF

			(* exitact *)
			IF eNewstep <>  E_FLM_CorkingStep.NoStep THEN
				;
			END_IF;
			
		(* Rotation *)
		E_FLM_CorkingStep.Rotation:
			(* entry action *)
			IF NOT bEntryact THEN
				bEntryact := TRUE;
			END_IF;

			(* body *)
			bErr := FALSE;
			
			bVertical := TRUE;
			bRotation := fbRotation.bRotation;			
			bRotationExecute := TRUE;					
							
			(* transition *)
			IF fbRotation.bError THEN
				eNewstep :=  E_FLM_CorkingStep.NeOrError;
			ELSE
				IF fbRotation.bDone THEN
					eNewstep :=  E_FLM_CorkingStep.Up;
				END_IF;			
			END_IF;

			(* exitact *)
			IF eNewstep <>  E_FLM_CorkingStep.NoStep THEN
				IF eNewstep = E_FLM_CorkingStep.NeOrError THEN
					eErrStep := E_FLM_CorkingStep.Rotation;
					nErrID := fbRotation.nErrId;
				END_IF
			END_IF;
			
		(* Up *)
		E_FLM_CorkingStep.Up:
			(* entry action *)
			IF NOT bEntryact THEN
				bEntryact := TRUE;
			END_IF;

			(* body *)
			bErr := FALSE;
			
			bVertical := TRUE;
			bRotation := FALSE;			
			bRotationExecute := FALSE;					
							
			(* transition *)
			IF tStepTime >= stParams.tUp THEN
				eNewstep :=  E_FLM_CorkingStep.Done;			
			END_IF;

			(* exitact *)
			IF eNewstep <>  E_FLM_CorkingStep.NoStep THEN
				;
			END_IF;
			
		(* Done *)
		E_FLM_CorkingStep.Done:
			(* entry action *)
			IF NOT bEntryact THEN
				bEntryact := TRUE;
			END_IF;

			(* body *)
			bErr := FALSE;
			
			bVertical := FALSE;
			bRotation := FALSE;			
			bRotationExecute := FALSE;					
							
			(* transition *)
			IF TRUE THEN
				eNewstep :=  E_FLM_CorkingStep.Ready;			
			END_IF;

			(* exitact *)
			IF eNewstep <>  E_FLM_CorkingStep.NoStep THEN
				;
			END_IF;			
					
		(* Stopping *)
		E_FLM_CorkingStep.Stopping:
			(* entry action *)
			IF NOT bEntryact THEN
				bEntryact := TRUE;
			END_IF;

			(* body *)
			bErr := FALSE;
			
			bVertical := FALSE;
			bRotation := FALSE;			
			bRotationExecute := FALSE;					
							
			(* transition *)
			IF TRUE THEN
				eNewstep :=  E_FLM_CorkingStep.Down;			
			END_IF;

			(* exitact *)
			IF eNewstep <>  E_FLM_CorkingStep.NoStep THEN
				;
			END_IF;	
		ELSE
			eNewstep :=  E_FLM_CorkingStep.NeOrError;
			eErrStep :=  E_FLM_CorkingStep.Unknown;			
			nErrID := 16#9999_9999;
	END_CASE
	
	(* call FBs *)	
	fbRotation(
		bExecute:= bRotationExecute, 
		bLimitSwitch:= bRotationLimitSwitch,	 
	);
	
	(* tempo di permanenza nello step *)
	fbTonStep(IN := (eNewstep =  E_FLM_CorkingStep.NoStep), PT := T#500H);
	tStepTime := fbTonStep.ET;
	
END_IF;

END_FUNCTION_BLOCK

// ---- FLM/Corking/FB_CorkingRotation.TcPOU
(* -----------------------------------------------------------------------------
| This sample has been supplied by Beckhoff As-Is and is intended only as an   |
| example implementation. Functionality is not guaranteed.                     |
----------------------------------------------------------------------------- *)

FUNCTION_BLOCK FB_CorkingRotation
VAR_INPUT
	bExecute : BOOL;
	bLimitSwitch : BOOL;
END_VAR
VAR_OUTPUT
	bRotation : BOOL; 
	bDone : BOOL;
	bError : BOOL;
	nErrId : UDINT;
END_VAR
VAR
	nCnt : UDINT;
END_VAR

(* -----------------------------------------------------------------------------
| This sample has been supplied by Beckhoff As-Is and is intended only as an   |
| example implementation. Functionality is not guaranteed.                     |
----------------------------------------------------------------------------- *)

IF bExecute THEN
	nCnt := nCnt + 1;
	bRotation := (nCnt >= 1 AND nCnt < 100) OR
				(nCnt >= 201 AND nCnt < 300) OR
				(nCnt >= 401 AND nCnt < 500) OR
				(nCnt >= 601 AND nCnt < 700) OR
				(nCnt >= 800 AND nCnt < 1000);
	IF nCnt >= 1000 THEN
		IF bLimitSwitch THEN
			bDone := TRUE;
			bError := FALSE;
			nErrId := 0;
		ELSE
			bDone := FALSE;
			bError := 1;
			nErrId := 16#9999_0001;
		END_IF			
	END_IF
ELSE
	bError := FALSE;
	bRotation := FALSE;
	nCnt := 0;
	bDone := FALSE;
END_IF

END_FUNCTION_BLOCK

// ---- FLM/FBs/FB_FLM_WriteOutputs.TcPOU
(* -----------------------------------------------------------------------------
| This sample has been supplied by Beckhoff As-Is and is intended only as an   |
| example implementation. Functionality is not guaranteed.                     |
----------------------------------------------------------------------------- *)

FUNCTION_BLOCK FB_FLM_WriteOutputs

VAR_INPUT
	stOut :  ST_FLM_Out;
	stParams : ST_FLM_Params;
END_VAR

VAR_IN_OUT
	stRawOut : ST_FLM_RawOut;	
END_VAR

VAR
	fbBlink : BLINK;
END_VAR

(* -----------------------------------------------------------------------------
| This sample has been supplied by Beckhoff As-Is and is intended only as an   |
| example implementation. Functionality is not guaranteed.                     |
----------------------------------------------------------------------------- *)

(* blinking *)
fbBlink(ENABLE:= TRUE, TIMELOW:= T#500MS, TIMEHIGH:= T#500MS);

(* lights and horn *)

IF stOut.bBlinkingYellow THEN
	stRawOut.bYellow := fbBlink.OUT;
ELSE
	IF stOut.bFixedYellow THEN
		stRawOut.bYellow := TRUE;
	ELSE
		stRawOut.bYellow := FALSE;
	END_IF
END_IF

IF stOut.bBlinkingGreen THEN
	stRawOut.bGreen := fbBlink.OUT;
ELSE
	IF stOut.bFixedGreen THEN
		stRawOut.bGreen := TRUE;
	ELSE
		stRawOut.bGreen := FALSE;
	END_IF
END_IF

stRawOut.bHorn := stOut.bHorn;

(* other digitals *)
stRawOut.bConveyor := stOut.bConveyor;
stRawOut.bWater := stOut.bWater;
stRawOut.bMint := stOut.bMint;
stRawOut.bCorkingVertical := stOut.bCorkingVertical;
stRawOut.bCorkingRotation := stOut.bCorkingRotation;

(*analogs *)

END_FUNCTION_BLOCK

// ---- POUs/SIMU_MAIN.TcPOU
(* -----------------------------------------------------------------------------
| This sample has been supplied by Beckhoff As-Is and is intended only as an   |
| example implementation. Functionality is not guaranteed.                     |
----------------------------------------------------------------------------- *)

PROGRAM SIMU_MAIN
VAR
	bInitialized : BOOL;
	fbVisuSim : FB_VisuSim;
	bRefillMint : BOOL;
	bRefillWater : BOOL;
	bEmergencyButton : BOOL;
	fPos : REAL;
END_VAR

(* -----------------------------------------------------------------------------
| This sample has been supplied by Beckhoff As-Is and is intended only as an   |
| example implementation. Functionality is not guaranteed.                     |
----------------------------------------------------------------------------- *)

IF NOT bInitialized THEN
	bEmergencyButton := TRUE;
	bInitialized := TRUE;
ELSE
	(* Visu and Simulation *)
	fbVisuSim(
		bConveyor := GVL_PLC.stFlmRawOut.bConveyor, 
		bWater := GVL_PLC.stFlmRawOut.bWater, 
		bMint := GVL_PLC.stFlmRawOut.bMint,
		bCorkingRotation := GVL_PLC.stFlmRawOut.bCorkingRotation, 
		bCokingVertical := GVL_PLC.stFlmRawOut.bCorkingVertical,
		bRefillWater := bRefillWater, 
		bRefillMint := bRefillMint,
		bEmergencyButton := bEmergencyButton,
	);
	fpos := fbVisuSim.fPos;
	GVL_PLC.stFlmRawIn.bEmergency := fbVisuSim.bEmergency;
	GVL_PLC.stFlmRawIn.bBottle := fbVisuSim.bBottle;
	GVL_PLC.stFlmRawIn.nWaterLevel := fbVisuSim.nWaterLevel;
	GVL_PLC.stFlmRawIn.nMintLevel := fbVisuSim.nMintLevel;
	GVL_PLC.stFlmRawIn.bCorkingRotationLimitSwitch := fbVisuSim.bCorkingRotationLimitSwitch; 
END_IF

END_PROGRAM

// ---- Simulation/FB_VisuSim.TcPOU
(* -----------------------------------------------------------------------------
| This sample has been supplied by Beckhoff As-Is and is intended only as an   |
| example implementation. Functionality is not guaranteed.                     |
----------------------------------------------------------------------------- *)

FUNCTION_BLOCK FB_VisuSim
VAR_INPUT
	bConveyor : BOOL;
	bWater : BOOL;
	bMint : BOOL;
	bCorkingRotation : BOOL;
	bCokingVertical : BOOL;
	bRefillWater : BOOL;
	bRefillMint : BOOL;
	bEmergencyButton : BOOL;
END_VAR
VAR_OUTPUT
	fPos : REAL;	
	bBottle : BOOL;
	nWaterLevel : INT;
	nMintLevel : INT;
	bCorkingRotationLimitSwitch : BOOL;
	bEmergency : BOOL;
END_VAR
VAR
	bInitialized : BOOL;	
	nCorkingRotationCnt : UINT;
	nCorkingRotationCntLowerLimit : UINT := 450;
END_VAR

(* -----------------------------------------------------------------------------
| This sample has been supplied by Beckhoff As-Is and is intended only as an   |
| example implementation. Functionality is not guaranteed.                     |
----------------------------------------------------------------------------- *)

IF NOT bInitialized THEN
	nWaterLevel := 32000;
	nMintLevel := 24000;
	bInitialized := TRUE;	
ELSE
	
	(* Simulazione pulsante di emergenza *)
	bEmergency := bEmergencyButton;	
	
	(* simulazione nastro trasportatore e sensore presenza bottiglia *)
	IF bConveyor THEN
		fPos := fPos + 0.1;
	END_IF
	
	IF fPos >= 120.0 THEN
		fPos := 0;
	END_IF
	
	bBottle := fPos >= 60.0 AND fPos <= 80.0;
	
	(* simulazione livelli acqua e menta *)
	IF bWater THEN
		nWaterLevel := nWaterLevel - 11;
	END_IF
	
	IF nWaterLevel < 0 THEN
		nWaterLevel := 0;
	END_IF
	
	IF bRefillWater THEN
		nWaterLevel := 31234;
	END_IF
	
	IF bMint THEN
		nMintLevel := nMintLevel - 17;
	END_IF
	
	IF nMintLevel < 0 THEN
		nMintLevel := 0;
	END_IF
	
	IF bRefillMint THEN
		nMintLevel := 28733;
	END_IF
	
	(* simulazione sensore tappatura *)
	IF bCokingVertical THEN
		IF bCorkingRotation THEN
			nCorkingRotationCnt := nCorkingRotationCnt + 1;
		END_IF
	ELSE
		nCorkingRotationCnt := 0;
	END_IF
	
	bCorkingRotationLimitSwitch := nCorkingRotationCnt > nCorkingRotationCntLowerLimit;
	
	
	
	
	
	
	
	
	
END_IF

END_FUNCTION_BLOCK

// ---- StateMachinePro/FB_StateMachinePro.TcPOU
FUNCTION_BLOCK FB_StateMachinePro
VAR_INPUT	
	bEnable : BOOL;
	bStart : BOOL;
	bStop : BOOL;
	
	bBottle : BOOL;				// fotocellula FC1
END_VAR

VAR_OUTPUT
	eStep :  E_Step;
	tStepTime : TIME;
	eErrStep : E_Step;
	nErrId : DINT;
	
	bConveyor : BOOL;			// nastro trasportatore
	bWater : BOOL;				// riempimento acqua
	bMint : BOOL;				// riempimento menta	
	bCorking : BOOL;			// inserimento del tappo	
END_VAR

VAR_IN_OUT
	
END_VAR

VAR
	bInitialized :  BOOL;
	eNewstep :  E_Step;
	bEntryact :  BOOL;
	fbTonStep :  TON;	
	
	fbTonBottle : TON;
	fbRtBottle : R_TRIG;
	
	fbRtStop : R_TRIG;
	bStopRequest : BOOL;
	
	nFillingCycles : USINT;
END_VAR

IF NOT bInitialized THEN
	eNewstep := E_Step.NoStep;
	eStep := E_Step.Stop;
	bEntryact := FALSE;
	bInitialized := TRUE;		
ELSE	
	(* disabilitata o avaria *)
	IF NOT bEnable THEN
		eNewstep := E_Step.NeOrError;
	END_IF;
	
	IF eNewstep <> E_Step.NoStep THEN
		eStep := eNewstep;
		eNewstep := E_Step.NoStep;
		bEntryact := FALSE;
	END_IF;

	(* filtri *)
	fbTonBottle(IN:= bBottle, PT:= T#500MS);		// filtro sensore presenza bottiglia
	
	(* fronti *)
	fbRtBottle(CLK:= fbTonBottle.Q);
	fbRtStop(CLK:= bStop);
	
	(* richieste *)
	IF fbRtStop.Q THEN
		bStopRequest := TRUE;
	END_IF; 
	
	CASE eStep OF
		
		(* not Enabled or Error *)
		E_Step.NeOrError :
			(* entry action *)
			IF NOT bEntryact THEN
				bEntryact := TRUE;
			END_IF;

			(* body *)
			bConveyor := FALSE;
			bWater := FALSE;
			bMint := FALSE;
			bCorking := FALSE;
			
			nFillingCycles := 0;
					
			(* transition *)
			IF bEnable THEN				
				eNewstep := E_Step.Stop;				
			END_IF;

			(* exitact *)
			IF eNewstep <> E_Step.NoStep THEN
				;
			END_IF;		
			
		(* Stop *)
		E_Step.Stop:
			(* entry action *)
			IF NOT bEntryact THEN
				bStopRequest := FALSE;
				bEntryact := TRUE;
			END_IF;

			(* body *)
			bConveyor := FALSE;
			bWater := FALSE;
			bMint := FALSE;
			bCorking := FALSE;
			
			nFillingCycles := 0;
				
			(* transition *)
			IF bStart THEN
				eNewstep := E_Step.Feeding;
			END_IF
			
			(* exitact *)
			IF eNewstep <> E_Step.NoStep THEN
				;
			END_IF;
			
		(* Feeding *)
		E_Step.Feeding:
			(* entry action *)
			IF NOT bEntryact THEN
				bEntryact := TRUE;
			END_IF;

			(* body *)
			bConveyor := TRUE;
			bWater := FALSE;
			bMint := FALSE;
			bCorking := FALSE;
		
			(* transition *)
			IF bStopRequest AND NOT bBottle THEN
				eNewstep := E_Step.Stopping;
			ELSE
				IF fbRtBottle.Q THEN
					eNewstep := E_Step.WaterFilling;
				END_IF
			END_IF
			
			(* exitact *)
			IF eNewstep <> E_Step.NoStep THEN
				;
			END_IF;
			
		(* Water Filling *)
		E_Step.WaterFilling:
			(* entry action *)
			IF NOT bEntryact THEN
				nFillingCycles := nFillingCycles + 1;
				bEntryact := TRUE;
			END_IF;

			(* body *)
			bConveyor := FALSE;
			bWater := TRUE;
			bMint := FALSE;
			bCorking := FALSE;
		
			(* transition *)
			IF tStepTime >= T#1S500MS THEN
				eNewstep := E_Step.MintFilling;
			END_IF
			
			(* exitact *)
			IF eNewstep <> E_Step.NoStep THEN
				;
			END_IF;
			
		(* Mint Filling *)
		E_Step.MintFilling:
			(* entry action *)
			IF NOT bEntryact THEN
				bEntryact := TRUE;
			END_IF;

			(* body *)
			bConveyor := FALSE;
			bWater := FALSE;
			bMint := TRUE;
			bCorking := FALSE;
		
			(* transition *)
			IF tStepTime >= T#500MS THEN
				IF nFillingCycles >= 3 THEN
					eNewstep := E_Step.Waiting1;
				ELSE 
					eNewstep := E_Step.WaterFilling;
				END_IF
					
			END_IF
			
			(* exitact *)
			IF eNewstep <> E_Step.NoStep THEN
				IF eNewstep = E_Step.Waiting1 THEN
					nFillingCycles := 0;
				END_IF
			END_IF;	

		(* Waiting 1 *)
		E_Step.Waiting1:
			(* entry action *)
			IF NOT bEntryact THEN
				bEntryact := TRUE;
			END_IF;

			(* body *)
			bConveyor := FALSE;
			bWater := FALSE;
			bMint := FALSE;
			bCorking := FALSE;
		
			(* transition *)
			IF tStepTime >= T#1S THEN
				eNewstep := E_Step.Corking;
			END_IF
			
			(* exitact *)
			IF eNewstep <> E_Step.NoStep THEN
				;
			END_IF;	

		(* Corking *)
		E_Step.Corking:
			(* entry action *)
			IF NOT bEntryact THEN
				bEntryact := TRUE;
			END_IF;

			(* body *)
			bConveyor := FALSE;
			bWater := FALSE;
			bMint := FALSE;
			bCorking := TRUE;
		
			(* transition *)
			IF tStepTime >= T#3S THEN
				eNewstep := E_Step.Waiting2;
			END_IF
			
			(* exitact *)
			IF eNewstep <> E_Step.NoStep THEN
				;
			END_IF;

		(* Waiting 2 *)
		E_Step.Waiting2:
			(* entry action *)
			IF NOT bEntryact THEN
				bEntryact := TRUE;
			END_IF;

			(* body *)
			bConveyor := FALSE;
			bWater := FALSE;
			bMint := FALSE;
			bCorking := FALSE;
		
			(* transition *)
			IF tStepTime >= T#1S THEN
				eNewstep := E_Step.Feeding;
			END_IF
			
			(* exitact *)
			IF eNewstep <> E_Step.NoStep THEN
				;
			END_IF;

		(* Stopping *)
		E_Step.Stopping:
			(* entry action *)
			IF NOT bEntryact THEN
				bEntryact := TRUE;
			END_IF;

			(* body *)
			bConveyor := FALSE;
			bWater := tStepTime >= T#200MS AND tStepTime <= T#400MS;
			bMint := tStepTime >= T#200MS AND tStepTime <= T#400MS;
			bCorking := FALSE;
		
			(* transition *)
			IF tStepTime >= T#2S THEN
				eNewstep := E_Step.Stop;
			END_IF; 
			
			(* exitact *)
			IF eNewstep <> E_Step.NoStep THEN
				;
			END_IF;		
		ELSE
			eNewstep := E_Step.NeOrError;
			eErrStep := E_Step.Unknown;
			nErrId := -9;			
	END_CASE;
	
	(* tempo di permanenza nello step *)
	fbTonStep(IN := (eNewstep = E_Step.NoStep), PT := T#500H);
	tStepTime := fbTonStep.ET;
	
END_IF;

END_FUNCTION_BLOCK

// ---- StateMachine/FB_StateMachine.TcPOU
(* -----------------------------------------------------------------------------
| This sample has been supplied by Beckhoff As-Is and is intended only as an   |
| example implementation. Functionality is not guaranteed.                     |
----------------------------------------------------------------------------- *)

FUNCTION_BLOCK FB_StateMachine
VAR_INPUT
	bStart : BOOL;
	bStop : BOOL;	
	bBottle : BOOL;				// fotocellula FC1	
END_VAR
VAR_OUTPUT
	bConveyor : BOOL;			// nastro trasportatore
	bWater : BOOL;				// riempimento acqua
	bMint : BOOL;				// riempimento menta	
	bCorking : BOOL;			// inserimento del tappo
END_VAR
VAR
	nStep : INT;
	
	fbTonBottle : TON;
	fbRtBottle : R_TRIG;
	
	fbTonStep2 : TON;
	fbTonStep3 : TON;
	fbTonStep4 : TON;
	fbTonStep5 : TON;
	fbTonStep6 : TON;
END_VAR

(* -----------------------------------------------------------------------------
| This sample has been supplied by Beckhoff As-Is and is intended only as an   |
| example implementation. Functionality is not guaranteed.                     |
----------------------------------------------------------------------------- *)

(* filtri *)
fbTonBottle(IN:= bBottle, PT:= T#500MS);		// filtro sensore presenza bottiglia

(* fronti *)
fbRtBottle(CLK:= fbTonBottle.Q);

(* tempo di permanenza negli step *)
fbTonStep2(IN:= nStep = 2, PT:= T#5S);			// tempo di riempimento acqua
fbTonStep3(IN:= nStep = 3, PT:= T#1S);			// tempo di riempimento menta
fbTonStep4(IN:= nStep = 4, PT:= T#1S);			// attesa prima di tappatura
fbTonStep5(IN:= nStep = 5, PT:= T#3S);			// tempo di tappatura
fbTonStep6(IN:= nStep = 6, PT:= T#1S);			// attesa dopo tappatura

CASE nStep OF
	0: (* macchina ferma *)
		bConveyor := FALSE;
		bWater := FALSE;
		bMint := FALSE;
		bCorking := FALSE;
		
		(* transition *)
		IF NOT bStop AND bStart THEN
			nStep := 1;
		END_IF
		
	1: (* avanzamento nastro *)
		bConveyor := TRUE;
		bWater := FALSE;
		bMint := FALSE;
		bCorking := FALSE;
		
		(* transition *)
		IF fbRtBottle.Q THEN
			nStep := 2;
		END_IF
		
	2: (* riempimento acqua *)
		bConveyor := FALSE;
		bWater := TRUE;
		bMint := FALSE;
		bCorking := FALSE;
		
		(* transition *)
		IF fbTonStep2.Q THEN
			nStep := 3;
		END_IF
		
	3: (* riempimento menta *)
		bConveyor := FALSE;
		bWater := FALSE;
		bMint := TRUE;
		bCorking := FALSE;
		
		(* transition *)
		IF fbTonStep3.Q THEN
			nStep := 4;
		END_IF
		
	4: (* attesa *)
		bConveyor := FALSE;
		bWater := FALSE;
		bMint := TRUE;
		bCorking := FALSE;
		
		(* transition *)
		IF fbTonStep4.Q THEN
			nStep := 5;
		END_IF
		
	5: (* tappatura *)
		bConveyor := FALSE;
		bWater := FALSE;
		bMint := FALSE;
		bCorking := TRUE;
		
		(* transition *)
		IF fbTonStep5.Q THEN
			nStep := 6;
		END_IF
		
	6: (* attesa *)
		bConveyor := FALSE;
		bWater := FALSE;
		bMint := FALSE;
		bCorking := FALSE;
		
		(* transition *)
		IF fbTonStep6.Q THEN
			nStep := 1;
		END_IF

END_CASE

END_FUNCTION_BLOCK

// ---- GlobalTextList.TcGTLO
TEXTLIST GlobalTextList
  663 = '%s'
  258 = 'ACK'
  899 = 'EMERGENCY'
  561 = 'FILLER MACHINE - FLM'
  475 = 'REFILL'
  445 = 'START'
  530 = 'STOP'
END_TEXTLIST

// ---- VISUs/Visu.TcVIS
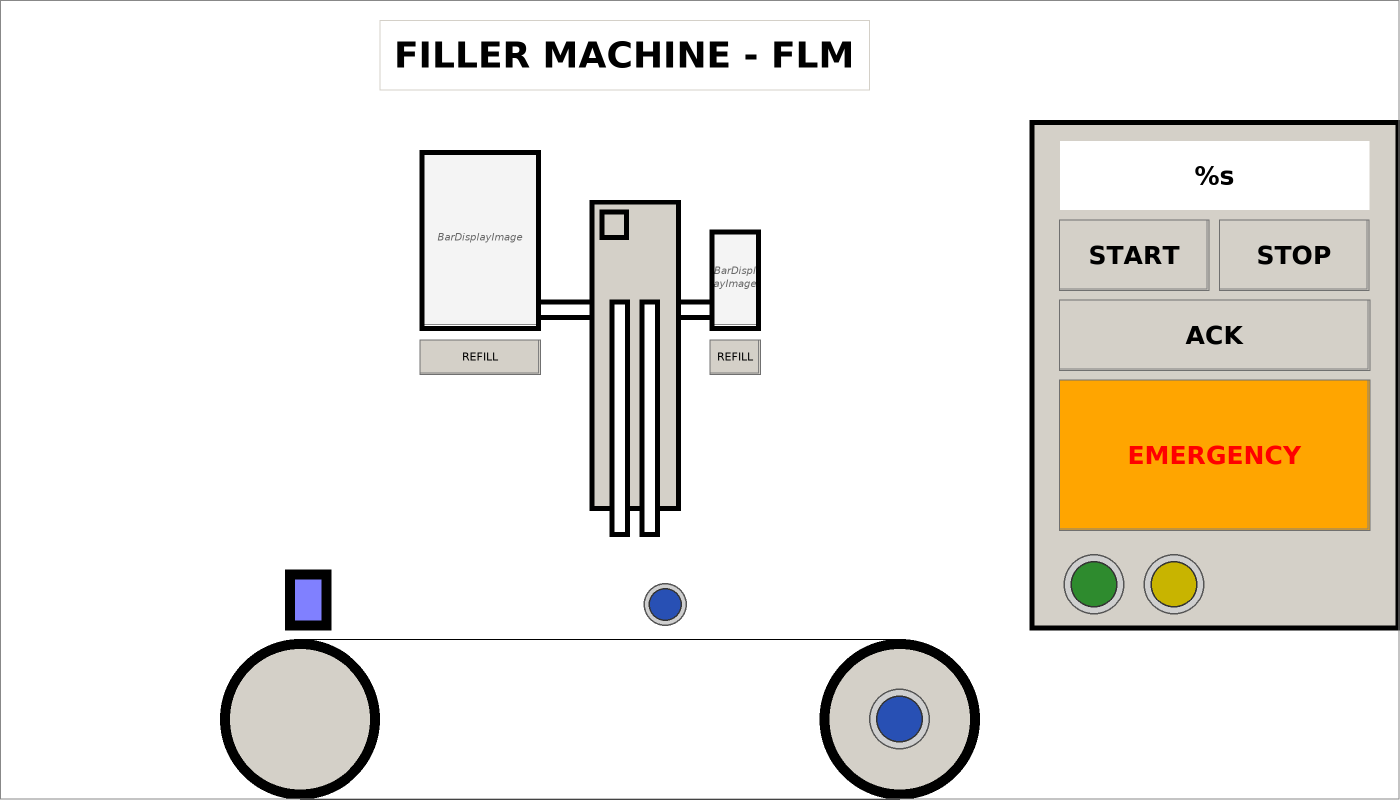
VISUALIZATION Visu  // 1401x801
    Rectangle (650,300 101x20), colour toggle: GVL_PLC.stFlmRawOut.bMint
    Rectangle (520,300 110x20), colour toggle: GVL_PLC.stFlmRawOut.bWater
    Rectangle (590,200 91x311), colour toggle: GVL_PLC.stFlmRawOut.bCorkingRotation
        p2738717112: (TO_REAL(GVL_PLC.stFlmRawOut.bCorkingVertical) * 50.0)
    Ellipse (220,640 160x160)
    Line (300,640) (900,640)
    Ellipse (820,640 160x160)
    Line (300,800) (900,800)
    Lamp1 (865,685 70x70), variable: GVL_PLC.stFlmRawOut.bConveyor, style: Lamp-Lamp1-Blue
    Rectangle (610,300 20x237), colour toggle: GVL_PLC.stFlmRawOut.bWater
    Rectangle (640,300 20x237), colour toggle: GVL_PLC.stFlmRawOut.bMint
    Lamp1 (640,580 51x50), variable: GVL_PLC.stFlmRawIn.bBottle, style: Lamp-Lamp1-Blue
    RoundedRectangle (285,570 46x61), invisible if: SIMU_MAIN.fPos > 100.0
        p3560616238: SIMU_MAIN.fPos * 5.0
    RoundedRectangle (1030,120 371x511)
    Button (1060,220 150x71), "START"
        tap GVL_PLC.stFlmRawIn.bStartButton
    Button (1220,220 150x71), "STOP"
        tap GVL_PLC.stFlmRawIn.bStopButton p1329445385=TRUE
    Textfield (1060,140 311x71), "%s", text variable: GVL_PLC.stFlmStatus.eStep
    Button (1060,300 311x71), "ACK"
        tap GVL_PLC.stFlmRawIn.bAckButton
    Button (1060,380 311x151), "EMERGENCY"
        toggle SIMU_MAIN.bEmergencyButton
    Group (710,230 51x101)
        BarDisplayImage (0,0 51x95), value: GVL_PLC.stFlmRawIn.nMintLevel, style: BarDisplayImage-Gray, scale format: %.1f, scale 0..32767
        Rectangle (0,0 51x101), colour toggle: GVL_PLC.stFlmRawOut.bCorkingRotation
    Group (420,150 121x181)
        BarDisplayImage (0,0 121x175), value: GVL_PLC.stFlmRawIn.nWaterLevel, style: BarDisplayImage-Gray, scale format: %.1f, scale 0..32767
        Rectangle (0,0 121x181), colour toggle: GVL_PLC.stFlmRawOut.bCorkingRotation
    RoundedRectangle (600,210 29x30), colour toggle: GVL_PLC.stFlmRawIn.bCorkingRotationLimitSwitch
        p2738717112: (TO_REAL(GVL_PLC.stFlmRawOut.bCorkingVertical) * 50.0)
    Button (420,340 121x35), "REFILL"
        tap SIMU_MAIN.bRefillWater
    Button (710,340 51x35), "REFILL"
        tap SIMU_MAIN.bRefillMint
    Lamp1 (1060,550 70x70), variable: GVL_PLC.stFlmRawOut.bGreen, style: Lamp-Lamp1-Green
    Lamp1 (1140,550 70x70), variable: GVL_PLC.stFlmRawOut.bYellow, style: Lamp-Lamp1-Yellow
    Textfield (380,20 490x70), "FILLER MACHINE - FLM"
END_VISUALIZATION
